{attribute 'pack_mode' := '1'}
TYPE U_JCL_Message :

UNION
	Cmd: T_JCL_Command;
	State: T_JCL_State;
	PrintDone: T_JCL_PrintDone;
	ReqCleaning: T_JCL_RequestCleaning;
	AlmMsg: T_JCL_AlmMsg;
END_UNION

END_TYPE

(* stored: Version 1.1.0.1, ProductVersion 3.1.0.25
   DUT U_JCL_Message: Id {e7fc896b-72c0-4aca-9062-419ca60938d0} *)
